// TIA Portal V19 export
TYPE "LEXCHANGETRAY_typeTrayCommands"
// stored: Access Published
   STRUCT
      trayType : Int;   // 0: 拘束托盘 1: 塑料托盘
      init : Bool;
   END_STRUCT;
END_TYPE
